FUNCTION_BLOCK eventToBool (* Basic Function Block Type *)
  (* Standard: 61499-2 *)
  (* Version 0.0, 16/01/2026, Schneider Electric, Template *)
  PACKAGE Hidryco.HidrycoLib;
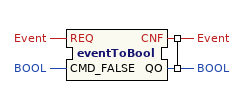
  EVENT_INPUT
    REQ; (* Normal Execution Request *)
  END_EVENT
  EVENT_OUTPUT
    CNF WITH QO; (* Execution Confirmation *)
  END_EVENT
  VAR_INPUT
    CMD_FALSE : BOOL;
  END_VAR
  VAR_OUTPUT
    QO : BOOL; (* Output event qualifier *)
  END_VAR
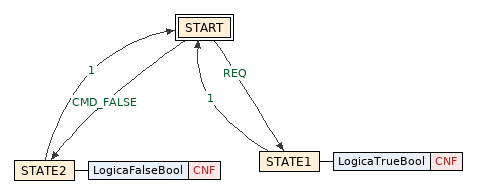
  EC_STATES
    START; (* Initial State *)
    STATE1 : LogicaTrueBool -> CNF;
    STATE2 : LogicaFalseBool -> CNF;
  END_STATES
  EC_TRANSITIONS
    START TO STATE1 := REQ;
    STATE1 TO START := 1;
    START TO STATE2 := CMD_FALSE;
    STATE2 TO START := 1;
  END_TRANSITIONS
  ALGORITHM LogicaTrueBool IN ST:
QO := TRUE;
;
  END_ALGORITHM
  ALGORITHM LogicaFalseBool IN ST:
QO := FALSE;
;
  END_ALGORITHM
END_FUNCTION_BLOCK
